INTERFACE ITF_Regelschuif

PROPERTY ActueelPosition : SINT
GET
END_GET
SET
END_SET
END_PROPERTY

METHOD RegelSchuifGoTo : SINT
VAR_INPUT
END_VAR
END_METHOD

PROPERTY StateRegelSchuif : E_RegelschuifState
GET
END_GET
SET
END_SET
END_PROPERTY

END_INTERFACE

(* stored: Version 1.1.0.1, ProductVersion 3.1.4026.8
   Itf ITF_Regelschuif: Id {5835ea1b-cb06-4d0c-8b0b-1d1de08323d4}
   Property ActueelPosition: Id {5d83e03f-02e3-4523-8fa3-9e754d6ad63b}
   Get Get: Id {e4b8c534-91c6-451c-baf1-f242802d57c7}
   Set Set: Id {b68299bb-4098-4290-9ff5-b5c633f37052}
   Method RegelSchuifGoTo: Id {99e424e3-8256-42ae-9d72-9807e7acbee4}
   Property StateRegelSchuif: Id {a07702d6-cb7e-47f4-a92d-65515d794b7e}
   Get Get: Id {3b94f187-ca1a-443e-b74f-f30c396f267c}
   Set Set: Id {bd4b0c98-c695-47b2-85e7-4f9d7b9d110c} *)
